FUNCTION_BLOCK Zone
  (* Version 1.0, 2006-11-13, Goran Cengic, Chalmers *)
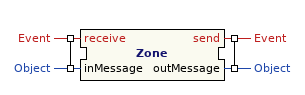
  EVENT_INPUT
    receive WITH inMessage;
  END_EVENT
  EVENT_OUTPUT
    send WITH outMessage;
  END_EVENT
  VAR_INPUT
    inMessage : Object;
  END_VAR
  VAR_OUTPUT
    outMessage : Object;
  END_VAR
END_FUNCTION_BLOCK
